ABB RobotStudio station: VRM_Rubik_v12.rspag

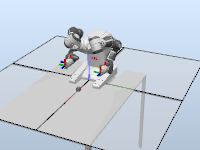
--- station ---
Station VRM_Rubik (saved by RobotStudio 20.4.9280.0)
Controller Controller_Rubik
  mechanical unit ROB_R: IRB14000_0.5_0.5_R, 6 joints, base frame (0, 0, 0) mm
  mechanical unit ROB_R_7: IRB14000_0.5_0.5_R, 1 joints, base frame (0, 0, 0) mm
  mechanical unit ROB_L: IRB14000_0.5_0.5_L, 6 joints, base frame (0, 0, 0) mm
  mechanical unit ROB_L_7: IRB14000_0.5_0.5_L, 1 joints, base frame (0, 0, 0) mm
Layout (positions relative to the parent item):
  - IRB14000_0.5_0.5 [mechanism, from Robots\IRB14000_0.5_0.5__02.rslib] at (0, 0, 0) mm
  - IRB14000_0.5_0.5_R [mechanism, from Robots\IRB14000_0.5_0.5__02.rslib] at (0, 0, 0) mm; joint values [0.0767, -2.326, -2.2629, 0.5469, 0.2972, 1.0609, -0.0992] (rad or m)
  - IRB14000_0.5_0.5_L [mechanism, from Robots\IRB14000_0.5_0.5__02.rslib] at (0, 0, 0) mm; joint values [-0.2847, -2.3545, 2.1434, 0.5675, 2.7327, -0.9321, -2.9148] (rad or m)
  - Smart_Gripper_Servo_Camera_Fingers [mechanism] at (35.8, -200, 200) mm, rotated rx 120.88 ry -90 rz 59.12 deg; joint values [0.025] (rad or m)
      TCP Servo at (0, 0, 114.2) mm
      TCP Camera at (-7.3, 28.3, 35.1) mm, rotated rx 0 ry 90 rz 90 deg
      links: HandBase, DownFinger, UpFinger, VacuumOne, VacuumTwo
  - Smart_Gripper_Servo_Fingers [mechanism] at (35.8, 200, 200) mm, rotated rx 169.62 ry -90 rz 10.38 deg; joint values [0.025] (rad or m)
      TCP Servo at (0, 0, 114.2) mm
      links: HandBase, DownFinger, UpFinger, VacuumOne, VacuumTwo
  - cube_1C3 [part] at (250, -19, 0) mm
  - cube_2C3 [part] at (250, -6, 0) mm
  - cube_3C3 [part] at (250, 7, 0) mm
  - cube_2C2 [part] at (237, -6, 0) mm
  - cube_1C2 [part] at (237, -19, 0) mm
  - cube_3C2 [part] at (237, 7, 0) mm
  - cube_2C1 [part] at (224, -6, 0) mm
  - cube_1C1 [part] at (224, -19, 0) mm
  - cube_3C1 [part] at (224, 7, 0) mm
  - cube_2B1 [part] at (224, -6, 13) mm
  - cube_1B1 [part] at (224, -19, 13) mm
  - cube_3B1 [part] at (224, 7, 13) mm
  - cube_1B2 [part] at (237, -19, 13) mm
  - cube_3B2 [part] at (237, 7, 13) mm
  - cube_2B3 [part] at (250, -6, 13) mm
  - cube_1B3 [part] at (250, -19, 13) mm
  - cube_3B3 [part] at (250, 7, 13) mm
  - core [part] at (243, 0, 19) mm
  - cube_2A3 [part] at (250, -6, 26) mm
  - cube_1A3 [part] at (250, -19, 26) mm
  - cube_3A3 [part] at (250, 7, 26) mm
  - cube_2A2 [part] at (237, -6, 26) mm
  - cube_1A2 [part] at (237, -19, 26) mm
  - cube_3A2 [part] at (237, 7, 26) mm
  - cube_2A1 [part] at (224, -6, 26) mm
  - cube_1A1 [part] at (224, -19, 26) mm
  - cube_3A1 [part] at (224, 7, 26) mm
  - Attacher_3C2 [smart component, from Components\Attacher.rslib]
      properties: Parent=core; Flange=0; Child=cube_3C2; Mount=false; Offset=[0 0 0]; Orientation=[0 0 0]
  - Attacher_1B1 [smart component, from Components\Attacher.rslib]
      properties: Parent=core; Flange=0; Child=cube_1B1; Mount=false; Offset=[0 0 0]; Orientation=[0 0 0]
  - Attacher_1B2 [smart component, from Components\Attacher.rslib]
      properties: Parent=core; Flange=0; Child=cube_1B2; Mount=false; Offset=[0 0 0]; Orientation=[0 0 0]
  - Attacher_1B3 [smart component, from Components\Attacher.rslib]
      properties: Parent=core; Flange=0; Child=cube_1B3; Mount=false; Offset=[0 0 0]; Orientation=[0 0 0]
  - Attacher_1C1 [smart component, from Components\Attacher.rslib]
      properties: Parent=core; Flange=0; Child=cube_1C1; Mount=false; Offset=[0 0 0]; Orientation=[0 0 0]
  - Attacher_1C2 [smart component, from Components\Attacher.rslib]
      properties: Parent=core; Flange=0; Child=cube_1C2; Mount=false; Offset=[0 0 0]; Orientation=[0 0 0]
  - Attacher_1C3 [smart component, from Components\Attacher.rslib]
      properties: Parent=core; Flange=0; Child=cube_1C3; Mount=false; Offset=[0 0 0]; Orientation=[0 0 0]
  - Attacher_2A1 [smart component, from Components\Attacher.rslib]
      properties: Parent=core; Flange=0; Child=cube_2A1; Mount=false; Offset=[0 0 0]; Orientation=[0 0 0]
  - Attacher_2A2 [smart component, from Components\Attacher.rslib]
      properties: Parent=core; Flange=0; Child=cube_2A2; Mount=false; Offset=[0 0 0]; Orientation=[0 0 0]
  - Attacher_2A3 [smart component, from Components\Attacher.rslib]
      properties: Parent=core; Flange=0; Child=cube_2A3; Mount=false; Offset=[0 0 0]; Orientation=[0 0 0]
  - Attacher_2B1 [smart component, from Components\Attacher.rslib]
      properties: Parent=core; Flange=0; Child=cube_2B1; Mount=false; Offset=[0 0 0]; Orientation=[0 0 0]
  - Attacher_2B3 [smart component, from Components\Attacher.rslib]
      properties: Parent=core; Flange=0; Child=cube_2B3; Mount=false; Offset=[0 0 0]; Orientation=[0 0 0]
  - Attacher_2C1 [smart component, from Components\Attacher.rslib]
      properties: Parent=core; Flange=0; Child=cube_2C1; Mount=false; Offset=[0 0 0]; Orientation=[0 0 0]
  - Attacher_2C2 [smart component, from Components\Attacher.rslib]
      properties: Parent=core; Flange=0; Child=cube_2C2; Mount=false; Offset=[0 0 0]; Orientation=[0 0 0]
  - Attacher_2C3 [smart component, from Components\Attacher.rslib]
      properties: Parent=core; Flange=0; Child=cube_2C3; Mount=false; Offset=[0 0 0]; Orientation=[0 0 0]
  - Attacher_3A1 [smart component, from Components\Attacher.rslib]
      properties: Parent=core; Flange=0; Child=cube_3A1; Mount=false; Offset=[0 0 0]; Orientation=[0 0 0]
  - Attacher_3A2 [smart component, from Components\Attacher.rslib]
      properties: Parent=core; Flange=0; Child=cube_3A2; Mount=false; Offset=[0 0 0]; Orientation=[0 0 0]
  - Attacher_3A3 [smart component, from Components\Attacher.rslib]
      properties: Parent=core; Flange=0; Child=cube_3A3; Mount=false; Offset=[0 0 0]; Orientation=[0 0 0]
  - Attacher_3B1 [smart component, from Components\Attacher.rslib]
      properties: Parent=core; Flange=0; Child=cube_3B1; Mount=false; Offset=[0 0 0]; Orientation=[0 0 0]
  - Attacher_3B2 [smart component, from Components\Attacher.rslib]
      properties: Parent=core; Flange=0; Child=cube_3B2; Mount=false; Offset=[0 0 0]; Orientation=[0 0 0]
  - Attacher_3B3 [smart component, from Components\Attacher.rslib]
      properties: Parent=core; Flange=0; Child=cube_3B3; Mount=false; Offset=[0 0 0]; Orientation=[0 0 0]
  - Attacher_3C1 [smart component, from Components\Attacher.rslib]
      properties: Parent=core; Flange=0; Child=cube_3C1; Mount=false; Offset=[0 0 0]; Orientation=[0 0 0]
  - Attacher_3C3 [smart component, from Components\Attacher.rslib]
      properties: Parent=core; Flange=0; Child=cube_3C3; Mount=false; Offset=[0 0 0]; Orientation=[0 0 0]
  - Attacher_1A3 [smart component, from Components\Attacher.rslib]
      properties: Parent=core; Flange=0; Child=cube_1A3; Mount=false; Offset=[0 0 0]; Orientation=[0 0 0]
  - Attacher_1A2 [smart component, from Components\Attacher.rslib]
      properties: Parent=core; Flange=0; Child=cube_1A2; Mount=false; Offset=[0 0 0]; Orientation=[0 0 0]
  - Attacher_1A1 [smart component, from Components\Attacher.rslib]
      properties: Parent=core; Flange=0; Child=cube_1A1; Mount=false; Offset=[0 0 0]; Orientation=[0 0 0]
  - Detacher_1A1 [smart component, from Components\Detacher.rslib]
      properties: Child=cube_1A1; KeepPosition=true
  - Detacher_1A2 [smart component, from Components\Detacher.rslib]
      properties: Child=cube_1A2; KeepPosition=true
  - Detacher_1A3 [smart component, from Components\Detacher.rslib]
      properties: Child=cube_1A3; KeepPosition=true
  - Detacher_1B1 [smart component, from Components\Detacher.rslib]
      properties: Child=cube_1B1; KeepPosition=true
  - Detacher_1B2 [smart component, from Components\Detacher.rslib]
      properties: Child=cube_1B2; KeepPosition=true
  - Detacher_1B3 [smart component, from Components\Detacher.rslib]
      properties: Child=cube_1B3; KeepPosition=true
  - Detacher_1C1 [smart component, from Components\Detacher.rslib]
      properties: Child=cube_1C1; KeepPosition=true
  - Detacher_1C2 [smart component, from Components\Detacher.rslib]
      properties: Child=cube_1C2; KeepPosition=true
  - Detacher_1C3 [smart component, from Components\Detacher.rslib]
      properties: Child=cube_1C3; KeepPosition=true
  - Detacher_2A1 [smart component, from Components\Detacher.rslib]
      properties: Child=cube_2A1; KeepPosition=true
  - Detacher_2A2 [smart component, from Components\Detacher.rslib]
      properties: Child=cube_2A2; KeepPosition=true
  - Detacher_2A3 [smart component, from Components\Detacher.rslib]
      properties: Child=cube_2A3; KeepPosition=true
  - Detacher_2B1 [smart component, from Components\Detacher.rslib]
      properties: Child=cube_2B1; KeepPosition=true
  - Detacher_2B3 [smart component, from Components\Detacher.rslib]
      properties: Child=cube_2B3; KeepPosition=true
  - Detacher_2C1 [smart component, from Components\Detacher.rslib]
      properties: Child=cube_2C1; KeepPosition=true
  - Detacher_2C2 [smart component, from Components\Detacher.rslib]
      properties: Child=cube_2C2; KeepPosition=true
  - Detacher_2C3 [smart component, from Components\Detacher.rslib]
      properties: Child=cube_2C3; KeepPosition=true
  - Detacher_3A1 [smart component, from Components\Detacher.rslib]
      properties: Child=cube_3A1; KeepPosition=true
  - Detacher_3A2 [smart component, from Components\Detacher.rslib]
      properties: Child=cube_3A2; KeepPosition=true
  - Detacher_3A3 [smart component, from Components\Detacher.rslib]
      properties: Child=cube_3A3; KeepPosition=true
  - Detacher_3B1 [smart component, from Components\Detacher.rslib]
      properties: Child=cube_3B1; KeepPosition=true
  - Detacher_3B2 [smart component, from Components\Detacher.rslib]
      properties: Child=cube_3B2; KeepPosition=true
  - Detacher_3B3 [smart component, from Components\Detacher.rslib]
      properties: Child=cube_3B3; KeepPosition=true
  - Detacher_3C1 [smart component, from Components\Detacher.rslib]
      properties: Child=cube_3C1; KeepPosition=true
  - Detacher_3C2 [smart component, from Components\Detacher.rslib]
      properties: Child=cube_3C2; KeepPosition=true
  - Detacher_3C3 [smart component, from Components\Detacher.rslib]
      properties: Child=cube_3C3; KeepPosition=true
  - Positioner_i1A1 [smart component, from Components\Positioner.rslib]
      properties: Object=cube_1A1; Position=[0.224 -0.019 0.026]; Orientation=[0 0 0]; Reference=Global; ReferenceObject=(none)
  - Positioner_i1A2 [smart component, from Components\Positioner.rslib]
      properties: Object=cube_1A2; Position=[0.237 -0.019 0.026]; Orientation=[0 0 0]; Reference=Global; ReferenceObject=(none)
  - Positioner_i1A3 [smart component, from Components\Positioner.rslib]
      properties: Object=cube_1A3; Position=[0.25 -0.019 0.026]; Orientation=[0 0 0]; Reference=Global; ReferenceObject=(none)
  - Positioner_i1B1 [smart component, from Components\Positioner.rslib]
      properties: Object=cube_1B1; Position=[0.224 -0.019 0.013]; Orientation=[0 0 0]; Reference=Global; ReferenceObject=(none)
  - Positioner_i1B2 [smart component, from Components\Positioner.rslib]
      properties: Object=cube_1B2; Position=[0.237 -0.019 0.013]; Orientation=[0 0 0]; Reference=Global; ReferenceObject=(none)
  - Positioner_i1B3 [smart component, from Components\Positioner.rslib]
      properties: Object=cube_1B3; Position=[0.25 -0.019 0.013]; Orientation=[0 0 0]; Reference=Global; ReferenceObject=(none)
  - Positioner_i1C1 [smart component, from Components\Positioner.rslib]
      properties: Object=cube_1C1; Position=[0.224 -0.019 0]; Orientation=[0 0 0]; Reference=Global; ReferenceObject=(none)
  - Positioner_i1C2 [smart component, from Components\Positioner.rslib]
      properties: Object=cube_1C2; Position=[0.237 -0.019 0]; Orientation=[0 0 0]; Reference=Global; ReferenceObject=(none)
  - Positioner_i1C3 [smart component, from Components\Positioner.rslib]
      properties: Object=cube_1C3; Position=[0.25 -0.019 0]; Orientation=[0 0 0]; Reference=Global; ReferenceObject=(none)
  - Positioner_i2A1 [smart component, from Components\Positioner.rslib]
      properties: Object=cube_2A1; Position=[0.224 -0.006 0.026]; Orientation=[0 0 0]; Reference=Global; ReferenceObject=(none)
  - Positioner_i2A2 [smart component, from Components\Positioner.rslib]
      properties: Object=cube_2A2; Position=[0.237 -0.006 0.026]; Orientation=[0 0 0]; Reference=Global; ReferenceObject=(none)
  - Positioner_i2A3 [smart component, from Components\Positioner.rslib]
      properties: Object=cube_2A3; Position=[0.25 -0.006 0.026]; Orientation=[0 0 0]; Reference=Global; ReferenceObject=(none)
  - Positioner_i2B1 [smart component, from Components\Positioner.rslib]
      properties: Object=cube_2B1; Position=[0.224 -0.006 0.013]; Orientation=[0 0 0]; Reference=Global; ReferenceObject=(none)
  - Positioner_i2B3 [smart component, from Components\Positioner.rslib]
      properties: Object=cube_2B3; Position=[0.25 -0.006 0.013]; Orientation=[0 0 0]; Reference=Global; ReferenceObject=(none)
  - Positioner_i2C1 [smart component, from Components\Positioner.rslib]
      properties: Object=cube_2C1; Position=[0.224 -0.006 0]; Orientation=[0 0 0]; Reference=Global; ReferenceObject=(none)
  - Positioner_i2C2 [smart component, from Components\Positioner.rslib]
      properties: Object=cube_2C2; Position=[0.237 -0.006 0]; Orientation=[0 0 0]; Reference=Global; ReferenceObject=(none)
  - Positioner_i2C3 [smart component, from Components\Positioner.rslib]
      properties: Object=cube_2C3; Position=[0.25 -0.006 0]; Orientation=[0 0 0]; Reference=Global; ReferenceObject=(none)
  - Positioner_i3A1 [smart component, from Components\Positioner.rslib]
      properties: Object=cube_3A1; Position=[0.224 0.007 0.026]; Orientation=[0 0 0]; Reference=Global; ReferenceObject=(none)
  - Positioner_i3A2 [smart component, from Components\Positioner.rslib]
      properties: Object=cube_3A2; Position=[0.237 0.007 0.026]; Orientation=[0 0 0]; Reference=Global; ReferenceObject=(none)
  - Positioner_i3A3 [smart component, from Components\Positioner.rslib]
      properties: Object=cube_3A3; Position=[0.25 0.007 0.026]; Orientation=[0 0 0]; Reference=Global; ReferenceObject=(none)
  - Positioner_i3B1 [smart component, from Components\Positioner.rslib]
      properties: Object=cube_3B1; Position=[0.224 0.007 0.013]; Orientation=[0 0 0]; Reference=Global; ReferenceObject=(none)
  - Positioner_i3B2 [smart component, from Components\Positioner.rslib]
      properties: Object=cube_3B2; Position=[0.237 0.007 0.013]; Orientation=[0 0 0]; Reference=Global; ReferenceObject=(none)
  - Positioner_i3B3 [smart component, from Components\Positioner.rslib]
      properties: Object=cube_3B3; Position=[0.25 0.007 0.013]; Orientation=[0 0 0]; Reference=Global; ReferenceObject=(none)
  - Positioner_i3C1 [smart component, from Components\Positioner.rslib]
      properties: Object=cube_3C1; Position=[0.224 0.007 0]; Orientation=[0 0 0]; Reference=Global; ReferenceObject=(none)
  - Positioner_i3C2 [smart component, from Components\Positioner.rslib]
      properties: Object=cube_3C2; Position=[0.237 0.007 0]; Orientation=[0 0 0]; Reference=Global; ReferenceObject=(none)
  - Positioner_i3C3 [smart component, from Components\Positioner.rslib]
      properties: Object=cube_3C3; Position=[0.25 0.007 0]; Orientation=[0 0 0]; Reference=Global; ReferenceObject=(none)
  - Positioner_iCORE [smart component, from Components\Positioner.rslib]
      properties: Object=core; Position=[0.243 0 0.019]; Orientation=[0 0 0]; Reference=Global; ReferenceObject=(none)
  - Positioner_rCORE [smart component, from Components\Positioner.rslib]
      properties: Object=core; Position=[0.25 0 0.2065]; Orientation=[-1.5707963267949 0 0]; Reference=Global; ReferenceObject=(none)
  - Positioner_r1A1 [smart component, from Components\Positioner.rslib] at (231, 7, 225) mm, rotated rx -90 ry 0 rz 0 deg
      properties: Object=cube_1A1; Position=[0.231 0.007 0.2255]; Orientation=[-1.5707963267949 0 0]; Reference=Global; ReferenceObject=(none)
  - Positioner_r1A2 [smart component, from Components\Positioner.rslib] at (244, 7, 225.5) mm, rotated rx -90 ry 0 rz 0 deg
      properties: Object=cube_1A2; Position=[0.244 0.007 0.2255]; Orientation=[-1.5707963267949 0 0]; Reference=Global; ReferenceObject=(none)
  - Positioner_r1A3 [smart component, from Components\Positioner.rslib] at (257, 7, 225.5) mm, rotated rx -90 ry 0 rz 0 deg
      properties: Object=cube_1A3; Position=[0.257 0.007 0.2255]; Orientation=[-1.5707963267949 0 0]; Reference=Global; ReferenceObject=(none)
  - Positioner_r1B1 [smart component, from Components\Positioner.rslib] at (231, -6, 225) mm, rotated rx -90 ry 0 rz 0 deg
      properties: Object=cube_1B1; Position=[0.231 -0.006 0.2255]; Orientation=[-1.5707963267949 0 0]; Reference=Global; ReferenceObject=(none)
  - Positioner_r1B2 [smart component, from Components\Positioner.rslib] at (244, -6, 225.5) mm, rotated rx -90 ry 0 rz 0 deg
      properties: Object=cube_1B2; Position=[0.244 -0.006 0.2255]; Orientation=[-1.5707963267949 0 0]; Reference=Global; ReferenceObject=(none)
  - Positioner_r1B3 [smart component, from Components\Positioner.rslib] at (257, -6, 225.5) mm, rotated rx -90 ry 0 rz 0 deg
      properties: Object=cube_1B3; Position=[0.257 -0.006 0.2255]; Orientation=[-1.5707963267949 0 0]; Reference=Global; ReferenceObject=(none)
  - Positioner_r1C1 [smart component, from Components\Positioner.rslib] at (231, -19, 225.5) mm, rotated rx -90 ry 0 rz 0 deg
      properties: Object=cube_1C1; Position=[0.231 -0.019 0.2255]; Orientation=[-1.5707963267949 0 0]; Reference=Global; ReferenceObject=(none)
  - Positioner_r1C2 [smart component, from Components\Positioner.rslib] at (244, -19, 225.5) mm, rotated rx -90 ry 0 rz 0 deg
      properties: Object=cube_1C2; Position=[0.244 -0.019 0.2255]; Orientation=[-1.5707963267949 0 0]; Reference=Global; ReferenceObject=(none)
  - Positioner_r1C3 [smart component, from Components\Positioner.rslib] at (257, -19, 225.5) mm, rotated rx -90 ry 0 rz 0 deg
      properties: Object=cube_1C3; Position=[0.257 -0.019 0.2255]; Orientation=[-1.5707963267949 0 0]; Reference=Global; ReferenceObject=(none)
  - Positioner_r2A1 [smart component, from Components\Positioner.rslib] at (231, 7, 212.5) mm, rotated rx -90 ry 0 rz 0 deg
      properties: Object=cube_2A1; Position=[0.231 0.007 0.2125]; Orientation=[-1.5707963267949 0 0]; Reference=Global; ReferenceObject=(none)
  - Positioner_r2A2 [smart component, from Components\Positioner.rslib] at (244, 7, 212.5) mm, rotated rx -90 ry 0 rz 0 deg
      properties: Object=cube_2A2; Position=[0.244 0.007 0.2125]; Orientation=[-1.5707963267949 0 0]; Reference=Global; ReferenceObject=(none)
  - Positioner_r2A3 [smart component, from Components\Positioner.rslib] at (257, 7, 212.5) mm, rotated rx -90 ry 0 rz 0 deg
      properties: Object=cube_2A3; Position=[0.257 0.007 0.2125]; Orientation=[-1.5707963267949 0 0]; Reference=Global; ReferenceObject=(none)
  - Positioner_r2B1 [smart component, from Components\Positioner.rslib] at (231, -6, 212.5) mm, rotated rx -90 ry 0 rz 0 deg
      properties: Object=cube_2B1; Position=[0.231 -0.006 0.2125]; Orientation=[-1.5707963267949 0 0]; Reference=Global; ReferenceObject=(none)
  - Positioner_r2B3 [smart component, from Components\Positioner.rslib] at (257, -6, 212.5) mm, rotated rx -90 ry 0 rz 0 deg
      properties: Object=cube_2B3; Position=[0.257 -0.006 0.2125]; Orientation=[-1.5707963267949 0 0]; Reference=Global; ReferenceObject=(none)
  - Positioner_r2C1 [smart component, from Components\Positioner.rslib] at (231, -19, 212.5) mm, rotated rx -90 ry 0 rz 0 deg
      properties: Object=cube_2C1; Position=[0.231 -0.019 0.2125]; Orientation=[-1.5707963267949 0 0]; Reference=Global; ReferenceObject=(none)
  - Positioner_r2C2 [smart component, from Components\Positioner.rslib] at (244, -19, 212.5) mm, rotated rx -90 ry 0 rz 0 deg
      properties: Object=cube_2C2; Position=[0.244 -0.019 0.2125]; Orientation=[-1.5707963267949 0 0]; Reference=Global; ReferenceObject=(none)
  - Positioner_r2C3 [smart component, from Components\Positioner.rslib] at (257, -19, 212.5) mm, rotated rx -90 ry 0 rz 0 deg
      properties: Object=cube_2C3; Position=[0.257 -0.019 0.2125]; Orientation=[-1.5707963267949 0 0]; Reference=Global; ReferenceObject=(none)
  - Positioner_r3A1 [smart component, from Components\Positioner.rslib] at (231, 7, 199.5) mm, rotated rx -90 ry 0 rz 0 deg
      properties: Object=cube_3A1; Position=[0.231 0.007 0.1995]; Orientation=[-1.5707963267949 0 0]; Reference=Global; ReferenceObject=(none)
  - Positioner_r3A2 [smart component, from Components\Positioner.rslib] at (244, 7, 199.5) mm, rotated rx -90 ry 0 rz 0 deg
      properties: Object=cube_3A2; Position=[0.244 0.007 0.1995]; Orientation=[-1.5707963267949 0 0]; Reference=Global; ReferenceObject=(none)
  - Positioner_r3A3 [smart component, from Components\Positioner.rslib] at (257, 7, 199.5) mm, rotated rx -90 ry 0 rz 0 deg
      properties: Object=cube_3A3; Position=[0.257 0.007 0.1995]; Orientation=[-1.5707963267949 0 0]; Reference=Global; ReferenceObject=(none)
  - Positioner_r3B1 [smart component, from Components\Positioner.rslib] at (231, -6, 199.5) mm, rotated rx -90 ry 0 rz 0 deg
      properties: Object=cube_3B1; Position=[0.231 -0.006 0.1995]; Orientation=[-1.5707963267949 0 0]; Reference=Global; ReferenceObject=(none)
  - Positioner_r3B2 [smart component, from Components\Positioner.rslib] at (244, -6, 199.5) mm, rotated rx -90 ry 0 rz 0 deg
      properties: Object=cube_3B2; Position=[0.244 -0.006 0.1995]; Orientation=[-1.5707963267949 0 0]; Reference=Global; ReferenceObject=(none)
  - Positioner_r3B3 [smart component, from Components\Positioner.rslib] at (257, -6, 199.5) mm, rotated rx -90 ry 0 rz 0 deg
      properties: Object=cube_3B3; Position=[0.257 -0.006 0.1995]; Orientation=[-1.5707963267949 0 0]; Reference=Global; ReferenceObject=(none)
  - Positioner_r3C1 [smart component, from Components\Positioner.rslib] at (231, -19, 199.5) mm, rotated rx -90 ry 0 rz 0 deg
      properties: Object=cube_3C1; Position=[0.231 -0.019 0.1995]; Orientation=[-1.5707963267949 0 0]; Reference=Global; ReferenceObject=(none)
  - Positioner_r3C2 [smart component, from Components\Positioner.rslib] at (244, -19, 199.5) mm, rotated rx -90 ry 0 rz 0 deg
      properties: Object=cube_3C2; Position=[0.244 -0.019 0.1995]; Orientation=[-1.5707963267949 0 0]; Reference=Global; ReferenceObject=(none)
  - Positioner_r3C3 [smart component, from Components\Positioner.rslib] at (257, -19, 199.5) mm, rotated rx -90 ry 0 rz 0 deg
      properties: Object=cube_3C3; Position=[0.257 -0.019 0.1995]; Orientation=[-1.5707963267949 0 0]; Reference=Global; ReferenceObject=(none)
  - table [part]
  - Attacher_L [smart component, from Components\Attacher.rslib]
      properties: Parent=Smart_Gripper_Servo_Fingers; Flange=0; Child=core; Mount=false; Offset=[0 0 0]; Orientation=[0 0 0]
  - Attacher_R [smart component, from Components\Attacher.rslib]
      properties: Parent=Smart_Gripper_Servo_Camera_Fingers; Flange=0; Child=core; Mount=false; Offset=[0 0 0]; Orientation=[0 0 0]
  - Detacher_core [smart component, from Components\Detacher.rslib]
      properties: Child=core; KeepPosition=true
Attachment: Smart_Gripper_Servo_Camera_Fingers is attached to IRB14000_0.5_0.5_R / Link7
Attachment: Smart_Gripper_Servo_Fingers is attached to IRB14000_0.5_0.5_L / Link7
EventTableEntry 3147: Group=, Trigger=DO_close_L 3148, Actions=[EventTableActionMechanicalPose 3149], Comment=, ActivationMode=2, Cyclic=false
EventTableTriggerIO 3148: IOValue=[1], IRC5Controller=? -1, Operator=0, SignalSource=Controller_Rubik 1733
EventTableActionMechanicalPose 3149: VirtualSignal=, Mechanism=Smart_Gripper_Servo_Fingers 1554, ToPoseName=SyncPosition, VirtualSignalValue=[1]
EventTableEntry 3164: Group=, Trigger=DO_close_R 3165, Actions=[EventTableActionMechanicalPose 3166], Comment=, ActivationMode=2, Cyclic=false
EventTableTriggerIO 3165: IOValue=[1], IRC5Controller=? -1, Operator=0, SignalSource=Controller_Rubik 1733
EventTableActionMechanicalPose 3166: VirtualSignal=, Mechanism=Smart_Gripper_Servo_Camera_Fingers 1546, ToPoseName=SyncPosition, VirtualSignalValue=[1]
EventTableEntry 3167: Group=, Trigger=DO_open_L 3168, Actions=[EventTableActionMechanicalPose 3169], Comment=, ActivationMode=2, Cyclic=false
EventTableTriggerIO 3168: IOValue=[1], IRC5Controller=? -1, Operator=0, SignalSource=Controller_Rubik 1733
EventTableActionMechanicalPose 3169: VirtualSignal=, Mechanism=Smart_Gripper_Servo_Fingers 1554, ToPoseName=HomePosition, VirtualSignalValue=[1]
EventTableEntry 3170: Group=, Trigger=DO_open_R 3171, Actions=[EventTableActionMechanicalPose 3172], Comment=, ActivationMode=2, Cyclic=false
EventTableTriggerIO 3171: IOValue=[1], IRC5Controller=? -1, Operator=0, SignalSource=Controller_Rubik 1733
EventTableActionMechanicalPose 3172: VirtualSignal=, Mechanism=Smart_Gripper_Servo_Camera_Fingers 1546, ToPoseName=HomePosition, VirtualSignalValue=[1]
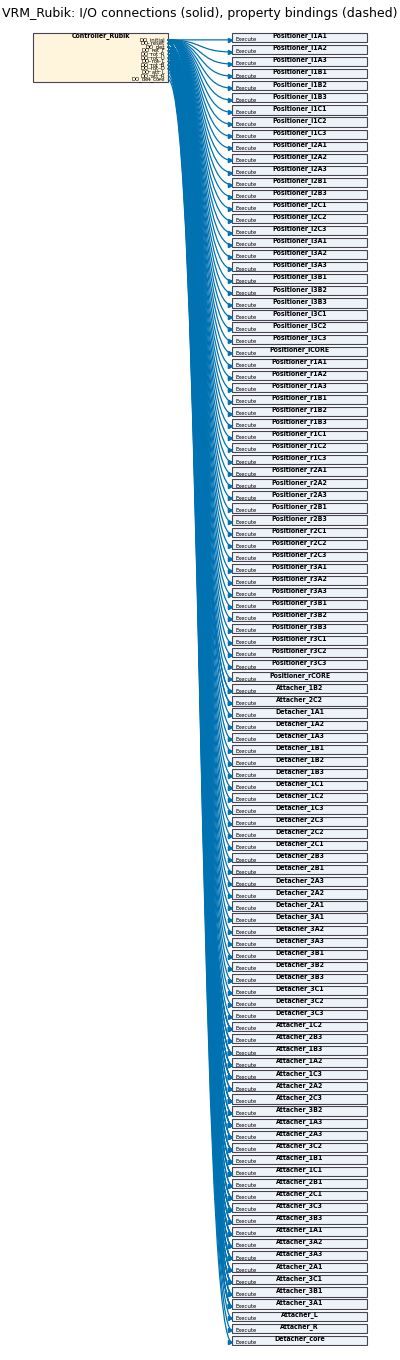
Station logic (signal -> signal, property => property):
  Controller_Rubik.DO_initial -> Positioner_i1A1.Execute
  Controller_Rubik.DO_initial -> Positioner_i1A2.Execute
  Controller_Rubik.DO_initial -> Positioner_i1A3.Execute
  Controller_Rubik.DO_initial -> Positioner_i1B1.Execute
  Controller_Rubik.DO_initial -> Positioner_i1B2.Execute
  Controller_Rubik.DO_initial -> Positioner_i1B3.Execute
  Controller_Rubik.DO_initial -> Positioner_i1C1.Execute
  Controller_Rubik.DO_initial -> Positioner_i1C2.Execute
  Controller_Rubik.DO_initial -> Positioner_i1C3.Execute
  Controller_Rubik.DO_initial -> Positioner_i2A1.Execute
  Controller_Rubik.DO_initial -> Positioner_i2A2.Execute
  Controller_Rubik.DO_initial -> Positioner_i2A3.Execute
  Controller_Rubik.DO_initial -> Positioner_i2B1.Execute
  Controller_Rubik.DO_initial -> Positioner_i2B3.Execute
  Controller_Rubik.DO_initial -> Positioner_i2C1.Execute
  Controller_Rubik.DO_initial -> Positioner_i2C2.Execute
  Controller_Rubik.DO_initial -> Positioner_i2C3.Execute
  Controller_Rubik.DO_initial -> Positioner_i3A1.Execute
  Controller_Rubik.DO_initial -> Positioner_i3A2.Execute
  Controller_Rubik.DO_initial -> Positioner_i3A3.Execute
  Controller_Rubik.DO_initial -> Positioner_i3B1.Execute
  Controller_Rubik.DO_initial -> Positioner_i3B2.Execute
  Controller_Rubik.DO_initial -> Positioner_i3B3.Execute
  Controller_Rubik.DO_initial -> Positioner_i3C1.Execute
  Controller_Rubik.DO_initial -> Positioner_i3C2.Execute
  Controller_Rubik.DO_initial -> Positioner_i3C3.Execute
  Controller_Rubik.DO_initial -> Positioner_iCORE.Execute
  Controller_Rubik.DO_reset -> Positioner_r1A1.Execute
  Controller_Rubik.DO_reset -> Positioner_r1A2.Execute
  Controller_Rubik.DO_reset -> Positioner_r1A3.Execute
  Controller_Rubik.DO_reset -> Positioner_r1B1.Execute
  Controller_Rubik.DO_reset -> Positioner_r1B2.Execute
  Controller_Rubik.DO_reset -> Positioner_r1B3.Execute
  Controller_Rubik.DO_reset -> Positioner_r1C1.Execute
  Controller_Rubik.DO_reset -> Positioner_r1C2.Execute
  Controller_Rubik.DO_reset -> Positioner_r1C3.Execute
  Controller_Rubik.DO_reset -> Positioner_r2A1.Execute
  Controller_Rubik.DO_reset -> Positioner_r2A2.Execute
  Controller_Rubik.DO_reset -> Positioner_r2A3.Execute
  Controller_Rubik.DO_reset -> Positioner_r2B1.Execute
  Controller_Rubik.DO_reset -> Positioner_r2B3.Execute
  Controller_Rubik.DO_reset -> Positioner_r2C1.Execute
  Controller_Rubik.DO_reset -> Positioner_r2C2.Execute
  Controller_Rubik.DO_reset -> Positioner_r2C3.Execute
  Controller_Rubik.DO_reset -> Positioner_r3A1.Execute
  Controller_Rubik.DO_reset -> Positioner_r3A2.Execute
  Controller_Rubik.DO_reset -> Positioner_r3A3.Execute
  Controller_Rubik.DO_reset -> Positioner_r3B1.Execute
  Controller_Rubik.DO_reset -> Positioner_r3B2.Execute
  Controller_Rubik.DO_reset -> Positioner_r3B3.Execute
  Controller_Rubik.DO_reset -> Positioner_r3C1.Execute
  Controller_Rubik.DO_reset -> Positioner_r3C2.Execute
  Controller_Rubik.DO_reset -> Positioner_r3C3.Execute
  Controller_Rubik.DO_reset -> Positioner_rCORE.Execute
  Controller_Rubik.DO_initial -> Attacher_1A1.Execute
  Controller_Rubik.DO_initial -> Attacher_1A2.Execute
  Controller_Rubik.DO_initial -> Attacher_1B1.Execute
  Controller_Rubik.DO_initial -> Attacher_1B2.Execute
  Controller_Rubik.DO_initial -> Attacher_1B3.Execute
  Controller_Rubik.DO_initial -> Attacher_1C1.Execute
  Controller_Rubik.DO_initial -> Attacher_1C2.Execute
  Controller_Rubik.DO_initial -> Attacher_1C3.Execute
  Controller_Rubik.DO_initial -> Attacher_2A1.Execute
  Controller_Rubik.DO_initial -> Attacher_2A2.Execute
  Controller_Rubik.DO_initial -> Attacher_2A3.Execute
  Controller_Rubik.DO_initial -> Attacher_2B1.Execute
  Controller_Rubik.DO_initial -> Attacher_2B3.Execute
  Controller_Rubik.DO_initial -> Attacher_2C1.Execute
  Controller_Rubik.DO_initial -> Attacher_2C2.Execute
  Controller_Rubik.DO_initial -> Attacher_2C3.Execute
  Controller_Rubik.DO_initial -> Attacher_3C3.Execute
  Controller_Rubik.DO_initial -> Attacher_3C2.Execute
  Controller_Rubik.DO_initial -> Attacher_3C1.Execute
  Controller_Rubik.DO_initial -> Attacher_3B3.Execute
  Controller_Rubik.DO_initial -> Attacher_3B2.Execute
  Controller_Rubik.DO_initial -> Attacher_3B1.Execute
  Controller_Rubik.DO_initial -> Attacher_3A3.Execute
  Controller_Rubik.DO_initial -> Attacher_3A2.Execute
  Controller_Rubik.DO_initial -> Attacher_3A1.Execute
  Controller_Rubik.DO_det -> Detacher_1A1.Execute
  Controller_Rubik.DO_det -> Detacher_1A2.Execute
  Controller_Rubik.DO_det -> Detacher_1A3.Execute
  Controller_Rubik.DO_det -> Detacher_1B1.Execute
  Controller_Rubik.DO_det -> Detacher_1B2.Execute
  Controller_Rubik.DO_det -> Detacher_1B3.Execute
  Controller_Rubik.DO_det -> Detacher_1C1.Execute
  Controller_Rubik.DO_det -> Detacher_1C2.Execute
  Controller_Rubik.DO_det -> Detacher_1C3.Execute
  Controller_Rubik.DO_det -> Detacher_2C3.Execute
  Controller_Rubik.DO_det -> Detacher_2C2.Execute
  Controller_Rubik.DO_det -> Detacher_2C1.Execute
  Controller_Rubik.DO_det -> Detacher_2B3.Execute
  Controller_Rubik.DO_det -> Detacher_2B1.Execute
  Controller_Rubik.DO_det -> Detacher_2A3.Execute
  Controller_Rubik.DO_det -> Detacher_2A2.Execute
  Controller_Rubik.DO_det -> Detacher_2A1.Execute
  Controller_Rubik.DO_det -> Detacher_3A1.Execute
  Controller_Rubik.DO_det -> Detacher_3A2.Execute
  Controller_Rubik.DO_det -> Detacher_3A3.Execute
  Controller_Rubik.DO_det -> Detacher_3B1.Execute
  Controller_Rubik.DO_det -> Detacher_3B2.Execute
  Controller_Rubik.DO_det -> Detacher_3B3.Execute
  Controller_Rubik.DO_det -> Detacher_3C1.Execute
  Controller_Rubik.DO_det -> Detacher_3C2.Execute
  Controller_Rubik.DO_det -> Detacher_3C3.Execute
  Controller_Rubik.DO_rot_F -> Attacher_1A1.Execute
  Controller_Rubik.DO_rot_F -> Attacher_1A2.Execute
  Controller_Rubik.DO_rot_F -> Attacher_1A3.Execute
  Controller_Rubik.DO_initial -> Attacher_1A3.Execute
  Controller_Rubik.DO_rot_F -> Attacher_1B1.Execute
  Controller_Rubik.DO_rot_F -> Attacher_1B2.Execute
  Controller_Rubik.DO_rot_F -> Attacher_1B3.Execute
  Controller_Rubik.DO_rot_F -> Attacher_1C1.Execute
  Controller_Rubik.DO_rot_F -> Attacher_1C2.Execute
  Controller_Rubik.DO_rot_F -> Attacher_1C3.Execute
  Controller_Rubik.DO_rot_R -> Attacher_1C1.Execute
  Controller_Rubik.DO_rot_R -> Attacher_1C2.Execute
  Controller_Rubik.DO_rot_R -> Attacher_1C3.Execute
  Controller_Rubik.DO_rot_R -> Attacher_2C1.Execute
  Controller_Rubik.DO_rot_R -> Attacher_2C2.Execute
  Controller_Rubik.DO_rot_R -> Attacher_2C3.Execute
  Controller_Rubik.DO_rot_R -> Attacher_3C1.Execute
  Controller_Rubik.DO_rot_R -> Attacher_3C2.Execute
  Controller_Rubik.DO_rot_R -> Attacher_3C3.Execute
  Controller_Rubik.DO_rot_U -> Attacher_1A3.Execute
  Controller_Rubik.DO_rot_U -> Attacher_1B3.Execute
  Controller_Rubik.DO_rot_U -> Attacher_1C3.Execute
  Controller_Rubik.DO_rot_U -> Attacher_2C3.Execute
  Controller_Rubik.DO_rot_U -> Attacher_2B3.Execute
  Controller_Rubik.DO_rot_U -> Attacher_2A3.Execute
  Controller_Rubik.DO_rot_U -> Attacher_3A3.Execute
  Controller_Rubik.DO_rot_U -> Attacher_3B3.Execute
  Controller_Rubik.DO_rot_U -> Attacher_3C3.Execute
  Controller_Rubik.DO_rot_L -> Attacher_1A1.Execute
  Controller_Rubik.DO_rot_L -> Attacher_1A2.Execute
  Controller_Rubik.DO_rot_L -> Attacher_1A3.Execute
  Controller_Rubik.DO_rot_L -> Attacher_2A1.Execute
  Controller_Rubik.DO_rot_L -> Attacher_2A2.Execute
  Controller_Rubik.DO_rot_L -> Attacher_2A3.Execute
  Controller_Rubik.DO_rot_L -> Attacher_3A1.Execute
  Controller_Rubik.DO_rot_L -> Attacher_3A2.Execute
  Controller_Rubik.DO_rot_L -> Attacher_3A3.Execute
  Controller_Rubik.DO_rot_B -> Attacher_3A1.Execute
  Controller_Rubik.DO_rot_B -> Attacher_3A2.Execute
  Controller_Rubik.DO_rot_B -> Attacher_3A3.Execute
  Controller_Rubik.DO_rot_B -> Attacher_3B1.Execute
  Controller_Rubik.DO_rot_B -> Attacher_3B2.Execute
  Controller_Rubik.DO_rot_B -> Attacher_3B3.Execute
  Controller_Rubik.DO_rot_B -> Attacher_3C1.Execute
  Controller_Rubik.DO_rot_B -> Attacher_3C2.Execute
  Controller_Rubik.DO_rot_B -> Attacher_3C3.Execute
  Controller_Rubik.DO_rot_D -> Attacher_1A1.Execute
  Controller_Rubik.DO_rot_D -> Attacher_2A1.Execute
  Controller_Rubik.DO_rot_D -> Attacher_3A1.Execute
  Controller_Rubik.DO_rot_D -> Attacher_1B1.Execute
  Controller_Rubik.DO_rot_D -> Attacher_2B1.Execute
  Controller_Rubik.DO_rot_D -> Attacher_3B1.Execute
  Controller_Rubik.DO_rot_D -> Attacher_1C1.Execute
  Controller_Rubik.DO_rot_D -> Attacher_2C1.Execute
  Controller_Rubik.DO_rot_D -> Attacher_3C1.Execute
  Controller_Rubik.DO_att_L -> Attacher_L.Execute
  Controller_Rubik.DO_att_R -> Attacher_R.Execute
  Controller_Rubik.DO_det_core -> Detacher_core.Execute
Targets, tools, work objects and paths stored in the station and not in the controller backup, written as RAPID:
! task T_ROB_R
MODULE Module1
  PROC Path_camera()
    MoveL Target_F_1,v1000,z100,Servo\WObj:=wobj0;
    MoveL Target_waiting,v1000,z100,Servo\WObj:=wobj0;
    MoveL Target_10,v1000,z100,Servo\WObj:=wobj0;
    MoveL Target_20,v1000,z100,Servo\WObj:=wobj0;
    MoveL Target_30,v1000,z100,Servo\WObj:=wobj0;
    MoveL Target_40,v1000,z100,Servo\WObj:=wobj0;
    MoveL Target_50,v1000,z100,Servo\WObj:=wobj0;
    MoveL Target_60,v1000,z100,Servo\WObj:=wobj0;
    MoveL Target_F,v1000,z100,Servo\WObj:=wobj0;
    MoveL Target_F_rot,v1000,z100,Servo\WObj:=wobj0;
    MoveL Target_home,v1000,z100,Servo\WObj:=wobj0;
    MoveL Target_R,v1000,z100,Servo\WObj:=wobj0;
    MoveL Target_R_rot,v1000,z100,Servo\WObj:=wobj0;
    MoveJ Target_home,v100,fine,Servo\WObj:=wobj0;
    MoveL Target_10,v100,fine,Servo\WObj:=wobj0;
    MoveJ Target_20,v100,fine,Servo\WObj:=wobj0;
    MoveL Target_30,v100,fine,Servo\WObj:=wobj0;
    MoveL Target_40,v100,fine,Servo\WObj:=wobj0;
    MoveL Target_50,v100,fine,Servo\WObj:=wobj0;
    MoveJ Target_60,v100,fine,Servo\WObj:=wobj0;
    MoveL Target_home,v100,fine,Servo\WObj:=wobj0;
    MoveL Target_F_1,v1000,z100,Servo\WObj:=wobj0;
    MoveL Target_F_1rot,v1000,z100,Servo\WObj:=wobj0;
    MoveL Target_B,v1000,z100,Servo\WObj:=wobj0;
    MoveL Target_D,v1000,z100,Servo\WObj:=wobj0;
    MoveL Target_U,v1000,z100,Servo\WObj:=wobj0;
  ENDPROC
ENDMODULE

! task T_ROB_L
MODULE Module1
  PROC Path_pick_up()
    MoveJ Target_10,v100,z100,Servo\WObj:=wobj0;
    MoveJ Target_20,v100,fine,Servo\WObj:=wobj0;
    MoveJ Target_waiting,v100,fine,Servo\WObj:=wobj0;
    MoveL Target_L,v1000,z100,Servo\WObj:=wobj0;
    MoveL Target_L_rot,v1000,z100,Servo\WObj:=wobj0;
    MoveL Target_B,v1000,z100,Servo\WObj:=wobj0;
    MoveL Target_B_rot,v1000,z100,Servo\WObj:=wobj0;
    MoveL Target_D,v1000,z100,Servo\WObj:=wobj0;
    MoveL Target_D_rot,v1000,z100,Servo\WObj:=wobj0;
    MoveL Target_U,v1000,z100,Servo\WObj:=wobj0;
    MoveL Target_U_rot,v1000,z100,Servo\WObj:=wobj0;
  ENDPROC
ENDMODULE


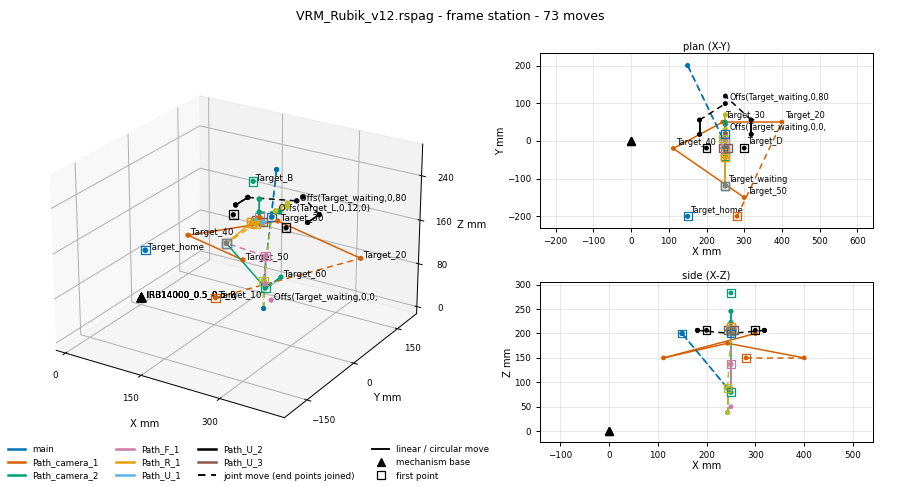
[picture p0: tool path of VRM_Rubik_v12.rspag in frame station, 73 of 73 moves have a stored position in this frame; points joined in program order, loops and branches not executed]
--- Backups/Controller_Rubik/RAPID/TASK1/PROGMOD/CalibData.mod ---
MODULE CalibData
    PERS tooldata Servo:=[TRUE,[[0,0,114.2],[1,0,0,0]],[0.229,[7.9,12.4,48.7],[1,0,0,0],0.00021,0.00023,0.00008]];
    PERS tooldata Camera:=[TRUE,[[-7.3,28.3,35.1],[0.5,-0.5,0.5,0.5]],[0.229,[7.9,12.4,48.7],[1,0,0,0],0.00021,0.00023,0.00008]];
ENDMODULE

--- Backups/Controller_Rubik/RAPID/TASK1/PROGMOD/Module1.mod ---
MODULE Module1
    CONST robtarget Target_10:=[[281,-200,150],[0.683012702,-0.183012702,0.683012702,-0.183012702],[0,0,1,4],[-101.964427132,9E+09,9E+09,9E+09,9E+09,9E+09]];
    CONST robtarget Target_20:=[[400,50,150],[0.612372436,-0.612372436,0.353553391,0.353553391],[1,-1,-1,4],[-101.964427132,9E+09,9E+09,9E+09,9E+09,9E+09]];
    CONST robtarget Target_30:=[[243,50,180],[0.707106781,-0.707106781,0,0],[1,-1,2,4],[-101.964427132,9E+09,9E+09,9E+09,9E+09,9E+09]];
    CONST robtarget Target_40:=[[112,-20,150],[0.612372436,-0.612372436,-0.353553391,-0.353553391],[0,-1,1,4],[-101.964427132,9E+09,9E+09,9E+09,9E+09,9E+09]];
    CONST robtarget Target_50:=[[300,-150,200],[0.707106781,0,0.707106781,0],[0,1,2,4],[-101.964427132,9E+09,9E+09,9E+09,9E+09,9E+09]];
    CONST robtarget Target_60:=[[250,50,80],[0,0,0.707106781,0.707106781],[1,-1,0,4],[-101.964427132,9E+09,9E+09,9E+09,9E+09,9E+09]];
    CONST robtarget Target_home:=[[150,-200,200],[0,0.707106781,0,0.707106781],[0,0,0,4],[-101.964427132,9E+09,9E+09,9E+09,9E+09,9E+09]];
    CONST robtarget Target_F:=[[250,0,225.5],[0,1,0,0],[-1,1,1,1],[-101.964421054,9E+09,9E+09,9E+09,9E+09,9E+09]];
    CONST robtarget Target_F_rot:=[[250,0,225.5],[0,-0.707106781,0.707106781,0],[-1,1,-2,1],[-101.964421054,9E+09,9E+09,9E+09,9E+09,9E+09]];
    CONST robtarget Target_R:=[[250,-19,206.5],[0.5,-0.5,-0.5,-0.5],[1,-1,1,4],[-101.964421054,9E+09,9E+09,9E+09,9E+09,9E+09]];
    CONST robtarget Target_R_rot:=[[250,-19,206.5],[0.707106781,-0.707106781,0,0],[1,-1,2,4],[-101.964421054,9E+09,9E+09,9E+09,9E+09,9E+09]];
    CONST robtarget Target_waiting:=[[250,-119,205],[0.5,-0.5,-0.5,-0.5],[1,-1,1,4],[-101.964421054,9E+09,9E+09,9E+09,9E+09,9E+09]];
    CONST robtarget Target_F_1:=[[250,0,75.5],[0,1,0,0],[1,2,-2,4],[-101.964421054,9E+09,9E+09,9E+09,9E+09,9E+09]];
    CONST robtarget Target_F_1rot:=[[250,0,75.5],[0,-0.707106781,0.707106781,0],[1,2,-1,4],[-101.964421054,9E+09,9E+09,9E+09,9E+09,9E+09]];
    CONST robtarget Target_B:=[[250,-39,283],[0.707106781,-0.707106781,0,0],[1,-1,-2,4],[-101.964421054,9E+09,9E+09,9E+09,9E+09,9E+09]];
    CONST robtarget Target_D:=[[300,-19,206.5],[0,0.707106781,0,0.707106781],[1,1,-1,4],[-101.964421054,9E+09,9E+09,9E+09,9E+09,9E+09]];
    CONST robtarget Target_U:=[[200,-19,206.5],[0.707106781,0,-0.707106781,0],[1,-1,1,4],[-101.964421054,9E+09,9E+09,9E+09,9E+09,9E+09]];

    PERS num state;
    PERS bool sync;
    VAR num state_R := 0;
    VAR socketdev serverSocket;
    VAR socketdev clientSocket;
    VAR string data;
    VAR string actualMove;
    VAR string dictionaryStr := "xxFRULBD";
    VAR num stringLen := 0;
    VAR num pos;

    PROC main()
        TEST state_R
            CASE 0: ! initial
                state := 2;
                Reset DO_rdy_L;
                Reset DO_rdy_R;
                PulseDO DO_det;
                PulseDO DO_det_core;
                PulseDO DO_initial;
                PulseDO DO_open_R;
                MoveJ Target_home,v100,fine,Servo\WObj:=wobj0;
                Path_camera_1;
                PulseDO DO_rdy_R;
                WaitDO DO_rdy_L, 1;
                Path_camera_2;
                PulseDO DO_rdy_R;
                state_R := 1;

            CASE 1: ! waiting for data
                SocketCreate serverSocket;
                SocketBind serverSocket, "127.0.0.1", 31254;
                SocketListen serverSocket;

                SocketAccept serverSocket, clientSocket, \Time:=WAIT_MAX;

                SocketReceive clientSocket \Str:=data;
                SocketSend clientSocket \Str:="recieved";

                SocketClose clientSocket;
                SocketClose serverSocket;

                stringLen := StrLen(data);

                IF stringLen <> 0  THEN
                    state_R := 2;
                ENDIF

            CASE 2: ! next move
                IF StrLen(data) = 0 THEN
                    WaitTime 2;
		            state := 10;
                    state_R := 10;
                ELSE
                    actualMove := StrPart(data, 1, 1);
                    data := StrPart(data, 2, stringLen-1);
                    stringLen := StrLen(data);
                    pos := StrFind(dictionaryStr, 1, actualMove);
		            state := pos;
                    state_R := pos;
                ENDIF

            CASE 3: ! F
                state := 9;
                WaitDO DO_rdy_L, 1;
                Path_F_1;
                PulseDO DO_rdy_R;
                state_R := 31;

            CASE 31:
                WaitDO DO_rdy_L, 1;
                state_R := 9;

            CASE 4: ! R
                state := 9;
                Path_R_1;
                PulseDO DO_rdy_R;
                state_R := 9;

            CASE 5: ! U
                state := 9;
                Path_U_1;
                PulseDO DO_rdy_R;
                state_R := 51;

            CASE 51:
                WaitDO DO_rdy_L, 1;
                Path_U_2;
                PulseDO DO_rdy_R;
                state_R := 52;

            CASE 52:
                WaitDO DO_rdy_L, 1;
                Path_U_3;
                PulseDO DO_rdy_R;
                state_R := 53;

            CASE 53:
                WaitDO DO_rdy_L, 1;
                Path_U_4;
                PulseDO DO_rdy_R;
                state_R := 9;

            CASE 6: ! L
                state := 9;
                Path_L_1;
                PulseDO DO_rdy_R;
                state_R := 61;

            CASE 61:
                WaitDO DO_rdy_L, 1;
                Path_L_2;
                state_R := 9;

            CASE 7: ! B
                state := 9;
                Path_B_1;
                PulseDO DO_rdy_R;
                state_R := 71;

            CASE 71:
                WaitDO DO_rdy_L, 1;
                Path_B_2;
                PulseDO DO_rdy_R;
                state_R := 72;

            CASE 72:
                WaitDO DO_rdy_L, 1;
                Path_B_3;
                PulseDO DO_rdy_R;
                state_R := 73;

            CASE 73:
                WaitDO DO_rdy_L, 1;
                Path_B_4;
                state_R := 9;

            CASE 8: ! D
                state := 9;
                Path_D_1;
                PulseDO DO_rdy_R;
                state_R := 81;

            CASE 81:
                WaitDO DO_rdy_L, 1;
                Path_D_2;
                PulseDO DO_rdy_R;
                state_R := 82;

            CASE 82:
                WaitDO DO_rdy_L, 1;
                Path_D_3;
                PulseDO DO_rdy_R;
                state_R := 83;

            CASE 83:
                WaitDO DO_rdy_L, 1;
                Path_D_4;
                PulseDO DO_rdy_R;
                state_R := 9;

            CASE 9:
                IF sync = TRUE THEN
                    state := 2;
                    state_R := 2;
                ENDIF

            CASE 10: ! end
                MoveJ Target_home,v100,fine,Servo\WObj:=wobj0;
                PulseDO DO_rdy_R;
        ENDTEST
    ENDPROC

    PROC Path_camera_1()
        MoveL Target_10,v100,fine,Servo\WObj:=wobj0;
        WaitTime 0.5;
        MoveJ Target_20,v100,fine,Servo\WObj:=wobj0;
        WaitTime 0.5;
        MoveL Target_30,v100,fine,Servo\WObj:=wobj0;
        WaitTime 0.5;
        MoveL Target_40,v100,fine,Servo\WObj:=wobj0;
        WaitTime 0.5;
        MoveL Target_50,v100,fine,Servo\WObj:=wobj0;
    ENDPROC

    PROC Path_camera_2()
        WaitTime 1;
        MoveJ Offs(Target_60, 0, -50, 0),v100,fine,Servo;
        MoveJ Target_60,v100,fine,Servo\WObj:=wobj0;
        WaitTime 0.5;
        MoveJ Offs(Target_60, 0, -50, 0),v100,fine,Servo;
        MoveL Target_waiting,v100,fine,Servo\WObj:=wobj0;
    ENDPROC

    PROC Path_F_1()
        MoveJ Offs(Target_F_1, 0, 0, 62),v100,z100,Servo;
        MoveL Offs(Target_F_1, 0, 0, 12),v100,fine,Servo;
        WaitTime 1;
        PulseDO DO_close_R;
        WaitTime 1;
        PulseDO DO_att_R;
        PulseDO DO_rot_F;
        MoveJ Offs(Target_F_1rot, 0, 0, 12),v100,fine,Servo;
        PulseDO DO_det;
        PulseDO DO_det_core;
        WaitTime 1;
        PulseDO DO_open_R;
        WaitTime 1;
        MoveJ Offs(Target_F_1rot, 0, 0, 62),v100,z100,Servo;
        MoveJ Target_waiting,v100,fine,Servo\WObj:=wobj0;
    ENDPROC

    PROC Path_R_1()
        MoveL Offs(Target_R, 0, -12, 0),v100,fine,Servo;
        WaitTime 1;
        PulseDO DO_close_R;
        WaitTime 1;
        PulseDO DO_att_R;
        PulseDO DO_rot_R;
        MoveJ Offs(Target_R_rot, 0, -12, 0),v100,fine,Servo;
        PulseDO DO_det;
        PulseDO DO_det_core;
        PulseDO DO_reset;
        WaitTime 1;
        PulseDO DO_open_R;
        WaitTime 1;
        MoveJ Target_waiting,v100,fine,Servo\WObj:=wobj0;
    ENDPROC

    PROC Path_U_1()
        MoveL Offs(Target_R, -6.5, 0, 0),v100,fine,Servo;
        WaitTime 1;
        PulseDO DO_close_R;
        WaitTime 1;
        PulseDO DO_att_R;
        PulseDO DO_rot_F;
        PulseDO DO_rot_R;
        PulseDO DO_rot_U;
        PulseDO DO_rot_L;
        PulseDO DO_rot_B;
        PulseDO DO_rot_D;
    ENDPROC

    PROC Path_U_2()
        MoveJ Target_U,v100,fine,Servo\WObj:=wobj0;
        PulseDO DO_det;
        PulseDO DO_det_core;
    ENDPROC

    PROC Path_U_3()
        PulseDO DO_att_R;
        PulseDO DO_rot_F;
        PulseDO DO_rot_R;
        PulseDO DO_rot_U;
        PulseDO DO_rot_L;
        PulseDO DO_rot_B;
        PulseDO DO_rot_D;
        MoveJ Offs(Target_R, -6.5, 0, 0),v100,fine,Servo;
        PulseDO DO_det;
        PulseDO DO_det_core;
        PulseDO DO_reset;
    ENDPROC

    PROC Path_U_4()
        WaitTime 3;
        PulseDO DO_open_R;
        WaitTime 1;
        MoveL Target_waiting,v100,fine,Servo\WObj:=wobj0;
    ENDPROC

    PROC Path_L_1()
        MoveL Target_R,v100,fine,Servo\WObj:=wobj0;
        WaitTime 1;
        PulseDO DO_close_R;
        WaitTime 1;
    ENDPROC

    PROC Path_L_2()
        WaitTime 1;
        PulseDO DO_open_R;
        WaitTime 1;
        MoveL Target_waiting,v100,fine,Servo\WObj:=wobj0;
    ENDPROC

    PROC Path_B_1()
        MoveL Offs(Target_R_rot, 0, -25, 6.5),v100,z100,Servo;
        MoveL Offs(Target_R_rot, 0, 0, 6.5),v100,fine,Servo;
        WaitTime 1;
        PulseDO DO_close_R;
        WaitTime 1;
        PulseDO DO_att_R;
        PulseDO DO_rot_F;
        PulseDO DO_rot_R;
        PulseDO DO_rot_U;
        PulseDO DO_rot_L;
        PulseDO DO_rot_B;
        PulseDO DO_rot_D;
    ENDPROC

    PROC Path_B_2()
        MoveJ Target_B,v100,fine,Servo\WObj:=wobj0;
        PulseDO DO_det;
        PulseDO DO_det_core;
    ENDPROC

    PROC Path_B_3()
        PulseDO DO_att_R;
        PulseDO DO_rot_F;
        PulseDO DO_rot_R;
        PulseDO DO_rot_U;
        PulseDO DO_rot_L;
        PulseDO DO_rot_B;
        PulseDO DO_rot_D;
        MoveJ Offs(Target_R_rot, 0, 0, 6.5),v100,fine,Servo;
        PulseDO DO_det;
        PulseDO DO_det_core;
        PulseDO DO_reset;
    ENDPROC

    PROC Path_B_4()
        WaitTime 1;
        PulseDO DO_open_R;
        WaitTime 1;
        MoveL Offs(Target_R_rot, 0, -25, 6.5),v100,z100,Servo;
        MoveL Target_waiting,v100,fine,Servo\WObj:=wobj0;
    ENDPROC

    PROC Path_D_1()
        MoveL Offs(Target_R, 6.5, 0, 0),v100,fine,Servo;
        WaitTime 1;
        PulseDO DO_close_R;
        WaitTime 1;
        PulseDO DO_att_R;
        PulseDO DO_rot_F;
        PulseDO DO_rot_R;
        PulseDO DO_rot_U;
        PulseDO DO_rot_L;
        PulseDO DO_rot_B;
        PulseDO DO_rot_D;
    ENDPROC

    PROC Path_D_2()
        MoveJ Target_D,v100,fine,Servo\WObj:=wobj0;
        PulseDO DO_det;
        PulseDO DO_det_core;
    ENDPROC

    PROC Path_D_3()
        PulseDO DO_att_R;
        PulseDO DO_rot_F;
        PulseDO DO_rot_R;
        PulseDO DO_rot_U;
        PulseDO DO_rot_L;
        PulseDO DO_rot_B;
        PulseDO DO_rot_D;
        MoveJ Offs(Target_R, 6.5, 0, 0),v100,fine,Servo;
        PulseDO DO_det;
        PulseDO DO_det_core;
        PulseDO DO_reset;
    ENDPROC

    PROC Path_D_4()
        WaitTime 1;
        PulseDO DO_open_R;
        WaitTime 1;
        MoveL Target_waiting,v100,fine,Servo\WObj:=wobj0;
    ENDPROC
ENDMODULE

--- Backups/Controller_Rubik/RAPID/TASK2/PROGMOD/CalibData.mod ---
MODULE CalibData
    PERS tooldata Servo:=[TRUE,[[0,0,114.2],[1,0,0,0]],[0.215,[8.7,12.3,49.2],[1,0,0,0],0.00021,0.00024,0.00009]];
ENDMODULE

--- Backups/Controller_Rubik/RAPID/TASK2/PROGMOD/Module1.mod ---
MODULE Module1
    CONST robtarget Target_10:=[[243,6.5,88],[0,1,0,0],[-1,-2,2,4],[101.964427132,9E+09,9E+09,9E+09,9E+09,9E+09]];
    CONST robtarget Target_20:=[[243,6.5,38],[0,1,0,0],[-1,-2,2,4],[101.964427132,9E+09,9E+09,9E+09,9E+09,9E+09]];
    CONST robtarget Target_waiting:=[[250,19,200],[0.707106781,0.707106781,0,0],[-1,1,-2,4],[101.964427132,9E+09,9E+09,9E+09,9E+09,9E+09]];
    CONST robtarget Target_home:=[[150,200,200],[0,0.707106781,0,0.707106781],[0,2,-2,5],[105.931421002,9E+09,9E+09,9E+09,9E+09,9E+09]];
    CONST robtarget Target_L:=[[250,19,206.5],[0.707106781,0.707106781,0,0],[-1,1,-2,4],[101.964427132,9E+09,9E+09,9E+09,9E+09,9E+09]];
    CONST robtarget Target_L_rot:=[[250,19,206.5],[0.5,0.5,-0.5,0.5],[-1,1,-2,4],[101.964427132,9E+09,9E+09,9E+09,9E+09,9E+09]];
    CONST robtarget Target_B:=[[250,-20,257.5],[0,0,0,1],[-1,0,0,4],[105.490331729,9E+09,9E+09,9E+09,9E+09,9E+09]];
    CONST robtarget Target_B_rot:=[[250,-20,257.5],[0.707106781,0,0,-0.707106781],[-1,0,0,4],[105.490331729,9E+09,9E+09,9E+09,9E+09,9E+09]];
    CONST robtarget Target_D:=[[318.5,5.5,206.5],[0.5,0.5,-0.5,0.5],[-1,1,-1,4],[101.964427132,9E+09,9E+09,9E+09,9E+09,9E+09]];
    CONST robtarget Target_D_rot:=[[318.5,5.5,206.5],[0,0,-0.707106781,0.707106781],[-1,1,-1,4],[101.964427132,9E+09,9E+09,9E+09,9E+09,9E+09]];
    CONST robtarget Target_U:=[[181.5,5.5,206.5],[0.5,0.5,-0.5,0.5],[0,1,-1,4],[105.931418404,9E+09,9E+09,9E+09,9E+09,9E+09]];
    CONST robtarget Target_U_rot:=[[181.5,5.5,206.5],[0,0,-0.707106781,0.707106781],[0,1,-1,4],[105.931418404,9E+09,9E+09,9E+09,9E+09,9E+09]];

    PERS num state;
    PERS bool sync;
    VAR num state_L := 0;

    PROC main()
        TEST state_L
            CASE 0: ! initial
                Reset DO_rdy_L;
                Reset DO_rdy_R;
                PulseDO DO_open_L;
                MoveJ Target_home,v100,fine,Servo\WObj:=wobj0;
                WaitDO DO_rdy_R, 1;
                Path_pick_up_1;
                PulseDO DO_rdy_L;
                WaitDO DO_rdy_R, 1;
                state_L := 2;

            CASE 2: ! next move
                sync := FALSE;
                state_L := state;

            CASE 3: ! F
                Path_F_1;
                PulseDO DO_rdy_L;
                state_L := 31;

            CASE 31:
                WaitDO DO_rdy_R, 1;
                Path_F_2;
                PulseDO DO_rdy_L;
                state_L := 2;

            CASE 4: ! R
                WaitDO DO_rdy_R, 1;
                state_L := 2;

            CASE 5: ! U
                WaitDO DO_rdy_R, 1;
                Path_U_1;
                PulseDO DO_rdy_L;
                state_L := 51;

            CASE 51:
                WaitDO DO_rdy_R, 1;
                Path_U_2;
                PulseDO DO_rdy_L;
                state_L := 52;

            CASE 52:
                WaitDO DO_rdy_R, 1;
                Path_U_3;
                PulseDO DO_rdy_L;
                state_L := 2;

            CASE 6: ! L
                WaitDO DO_rdy_R, 1;
                Path_L_1;
                PulseDO DO_rdy_L;
                state_L := 2;

            CASE 7: ! B
                WaitDO DO_rdy_R, 1;
                Path_B_1;
                PulseDO DO_rdy_L;
                state_L := 71;

            CASE 71:
                WaitDO DO_rdy_R, 1;
                Path_B_2;
                PulseDO DO_rdy_L;
                state_L := 72;

            CASE 72:
                WaitDO DO_rdy_R, 1;
                Path_B_3;
                PulseDO DO_rdy_L;
                state_L := 2;

            CASE 8: ! D
                WaitDO DO_rdy_R, 1;
                Path_D_1;
                PulseDO DO_rdy_L;
                state_L := 81;

            CASE 81:
                WaitDO DO_rdy_R, 1;
                Path_D_2;
                PulseDO DO_rdy_L;
                state_L := 82;

            CASE 82:
                WaitDO DO_rdy_R, 1;
                Path_D_3;
                PulseDO DO_rdy_L;
                state_L := 2;

            CASE 9:
                sync := TRUE;
                state_L := state;

            CASE 10: ! end
                WaitDO DO_rdy_R, 1;
                PulseDO DO_att_L;
                PulseDO DO_rot_F;
                PulseDO DO_rot_R;
                PulseDO DO_rot_U;
                PulseDO DO_rot_L;
                PulseDO DO_rot_B;
                PulseDO DO_rot_D;
                MoveJ Target_10,v100,z100,Servo\WObj:=wobj0;
                MoveJ Target_20,v100,fine,Servo\WObj:=wobj0;
                PulseDO DO_det;
                PulseDO DO_det_core;
                WaitTime 1;
                PulseDO DO_open_L;
                WaitTime 1;
                MoveJ Target_10,v100,z100,Servo\WObj:=wobj0;
                MoveJ Target_home,v100,fine,Servo\WObj:=wobj0;
                EXIT;
        ENDTEST
    ENDPROC

    PROC Path_pick_up_1()
        MoveJ Target_10,v100,z100,Servo\WObj:=wobj0;
        MoveJ Target_20,v100,fine,Servo\WObj:=wobj0;
        PulseDO DO_att_L;
        WaitTime 1;
        PulseDO DO_close_L;
        WaitTime 1;
        MoveJ Target_10,v100,z100,Servo\WObj:=wobj0;
        MoveJ Target_waiting,v100,fine,Servo\WObj:=wobj0;
        PulseDO DO_det;
        PulseDO DO_det_core;
    ENDPROC

    PROC Path_F_1()
        PulseDO DO_att_L;
        PulseDO DO_rot_F;
        PulseDO DO_rot_R;
        PulseDO DO_rot_U;
        PulseDO DO_rot_L;
        PulseDO DO_rot_B;
        PulseDO DO_rot_D;
        MoveL Offs(Target_waiting, 0, 0, -150),v100,fine,Servo;
        PulseDO DO_det;
        PulseDO DO_det_core;
    ENDPROC

    PROC Path_F_2()
        PulseDO DO_att_L;
        PulseDO DO_rot_F;
        PulseDO DO_rot_R;
        PulseDO DO_rot_U;
        PulseDO DO_rot_L;
        PulseDO DO_rot_B;
        PulseDO DO_rot_D;
        MoveL Target_waiting,v100,fine,Servo\WObj:=wobj0;
        PulseDO DO_det;
        PulseDO DO_det_core;
        PulseDO DO_reset;
    ENDPROC

    PROC Path_U_1()
        WaitTime 3;
        PulseDO DO_open_L;
        WaitTime 1;
        MoveL Offs(Target_waiting, 0, 80, 0),v100,fine,Servo;
    ENDPROC

    PROC Path_U_2()
        MoveJ Offs(Target_U, 0, 50, 0),v100,z100,Servo;
        MoveL Offs(Target_U, 0, 12, 0),v100,fine,Servo;
        WaitTime 1;
        PulseDO DO_close_L;
        WaitTime 1;
        PulseDO DO_att_L;
        PulseDO DO_rot_U;
        MoveJ Offs(Target_U_rot, 0, 12, 0),v100,fine,Servo;
        PulseDO DO_det;
        PulseDO DO_det_core;
        WaitTime 1;
        PulseDO DO_open_L;
        WaitTime 1;
        MoveL Offs(Target_U, 0, 50, 0),v100,z100,Servo;
        MoveJ Offs(Target_waiting, 0, 80, 0),v100,fine,Servo;
    ENDPROC

    PROC Path_U_3()
        MoveL Target_waiting,v100,fine,Servo\WObj:=wobj0;
        WaitTime 1;
        PulseDO DO_close_L;
        WaitTime 1;
    ENDPROC

    PROC Path_L_1()
        WaitTime 3;
        PulseDO DO_open_L;
        WaitTime 1;
        MoveL Offs(Target_L, 0, 50, 0),v100,z100,Servo;
        MoveL Offs(Target_L, 0, 12, 0),v100,fine,Servo;
        WaitTime 1;
        PulseDO DO_close_L;
        WaitTime 1;
        PulseDO DO_att_L;
        PulseDO DO_rot_L;
        MoveJ Offs(Target_L_rot, 0, 12, 0),v100,fine,Servo;
        PulseDO DO_det;
        PulseDO DO_det_core;
        PulseDO DO_reset;
        WaitTime 1;
        PulseDO DO_open_L;
        WaitTime 1;
        MoveL Offs(Target_L_rot, 0, 50, 0),v100,z100,Servo;
        MoveJ Offs(Target_waiting, 0, 50, 0),v100,fine,Servo;
        MoveL Target_waiting,v100,fine,Servo\WObj:=wobj0;
        WaitTime 1;
        PulseDO DO_close_L;
        WaitTime 1;
    ENDPROC

    PROC Path_B_1()
        WaitTime 3;
        PulseDO DO_open_L;
        WaitTime 1;
        MoveL Offs(Target_waiting, 0, 25, 0),v100,fine,Servo;
    ENDPROC

    PROC Path_B_2()
        MoveJ Offs(Target_B, 0, 0, -35),v100,z100,Servo;
        MoveL Offs(Target_B, 0, 0, -12),v100,fine,Servo;
        WaitTime 1;
        PulseDO DO_close_L;
        WaitTime 1;
        PulseDO DO_att_L;
        PulseDO DO_rot_B;
        MoveJ Offs(Target_B_rot, 0, 0, -12),v100,fine,Servo;
        PulseDO DO_det;
        PulseDO DO_det_core;
        WaitTime 1;
        PulseDO DO_open_L;
        WaitTime 1;
        MoveL Offs(Target_B_rot, 0, 0, -35),v100,z100,Servo;
        MoveJ Offs(Target_waiting, 0, 25, 0),v100,fine,Servo;
    ENDPROC

    PROC Path_B_3()
        MoveL Target_waiting,v100,fine,Servo\WObj:=wobj0;
        WaitTime 1;
        PulseDO DO_close_L;
        WaitTime 1;
    ENDPROC

    PROC Path_D_1()
        WaitTime 3;
        PulseDO DO_open_L;
        WaitTime 1;
        MoveL Offs(Target_waiting, 0, 100, 0),v100,fine,Servo;
    ENDPROC

    PROC Path_D_2()
        MoveJ Offs(Target_D, 0, 50, 0),v100,z100,Servo;
        MoveL Offs(Target_D, 0, 12, 0),v100,fine,Servo;
        WaitTime 1;
        PulseDO DO_close_L;
        WaitTime 1;
        PulseDO DO_att_L;
        PulseDO DO_rot_D;
        MoveL Offs(Target_D_rot, 0, 12, 0),v100,fine,Servo;
        PulseDO DO_det;
        PulseDO DO_det_core;
        WaitTime 1;
        PulseDO DO_open_L;
        WaitTime 1;
        MoveL Offs(Target_D, 0, 50, 0),v100,z100,Servo;
        MoveJ Offs(Target_waiting, 0, 100, 0),v100,fine,Servo;
    ENDPROC

    PROC Path_D_3()
        MoveL Target_waiting,v100,fine,Servo\WObj:=wobj0;
        WaitTime 1;
        PulseDO DO_close_L;
        WaitTime 1;
    ENDPROC
ENDMODULE

--- Backups/Controller_Rubik/SYSPAR/EIO.cfg ---
EIO:CFG_1.0:6:1::
#
SYSSIG_IN:

      -Signal "Collision_Avoidance" -Action "CollAvoidance"
#
INDUSTRIAL_NETWORK:

      -Name "EtherNetIP" -Connection "Private Network"\
      -Label "EtherNet/IP Adapter Network"

      -Name "DeviceNet" -Label "DeviceNet Master/Slave Network" -Address "2"
#
EIO_CROSS:

      -Name "Cross_Signal_Lamp" -Res "Signal_Lamp" -Act1 "DRV1BRAKE"
#
EIO_SIGNAL_SAFELEVEL:

      -Name "FlangePowerSafeLevel" -ActionWhenStartup "Last"
#
DEVICENET_DEVICE:

      -Name "D652_10" -VendorName "ABB Robotics" -ProductName "24 VDC Unit"\
      -Address 10 -ProductCode 26 -DeviceType 7 -ConnectionType "COS"\
      -OutputSize 2 -InputSize 2
#
DEVICENET_INTERNAL_DEVICE:

      -Name "DN_Internal_Device" -VendorName "ABB Robotics"\
      -ProductName "DeviceNet Internal Slave Device"
#
ETHERNETIP_INTERNAL_DEVICE:

      -Name "EN_Internal_Device" -VendorName "ABB Robotics"\
      -ProductName "EtherNet/IP Internal Adapter Device"
#
EIO_SIGNAL:

      -Name "custom_DI_0" -SignalType "DI" -Device "D652_10" -DeviceMap "0"

      -Name "custom_DI_1" -SignalType "DI" -Device "D652_10" -DeviceMap "1"

      -Name "custom_DI_2" -SignalType "DI" -Device "D652_10" -DeviceMap "2"

      -Name "custom_DI_3" -SignalType "DI" -Device "D652_10" -DeviceMap "3"

      -Name "custom_DI_4" -SignalType "DI" -Device "D652_10" -DeviceMap "4"

      -Name "custom_DI_5" -SignalType "DI" -Device "D652_10" -DeviceMap "5"

      -Name "custom_DI_6" -SignalType "DI" -Device "D652_10" -DeviceMap "6"

      -Name "custom_DI_7" -SignalType "DI" -Device "D652_10" -DeviceMap "7"

      -Name "custom_DO_0" -SignalType "DO" -Device "D652_10" -DeviceMap "0"

      -Name "custom_DO_1" -SignalType "DO" -Device "D652_10" -DeviceMap "1"

      -Name "custom_DO_2" -SignalType "DO" -Device "D652_10" -DeviceMap "2"

      -Name "custom_DO_3" -SignalType "DO" -Device "D652_10" -DeviceMap "3"

      -Name "custom_DO_4" -SignalType "DO" -Device "D652_10" -DeviceMap "4"

      -Name "custom_DO_5" -SignalType "DO" -Device "D652_10" -DeviceMap "5"

      -Name "custom_DO_6" -SignalType "DO" -Device "D652_10" -DeviceMap "6"

      -Name "custom_DO_7" -SignalType "DO" -Device "D652_10" -DeviceMap "7"

      -Name "hall_sensor_joint_1" -SignalType "DI" -Device "D652_10"\
      -DeviceMap "8"

      -Name "hall_sensor_joint_2" -SignalType "DI" -Device "D652_10"\
      -DeviceMap "9"

      -Name "hall_sensor_joint_3" -SignalType "DI" -Device "D652_10"\
      -DeviceMap "11"

      -Name "hall_sensor_joint_4" -SignalType "DI" -Device "D652_10"\
      -DeviceMap "12"

      -Name "hall_sensor_joint_5" -SignalType "DI" -Device "D652_10"\
      -DeviceMap "13"

      -Name "hall_sensor_joint_6" -SignalType "DI" -Device "D652_10"\
      -DeviceMap "14"

      -Name "hall_sensor_joint_7" -SignalType "DI" -Device "D652_10"\
      -DeviceMap "10"

      -Name "hall_sensor_24V_ROB_R" -SignalType "DO" -Device "D652_10"\
      -DeviceMap "8"

      -Name "hall_sensor_24V_ROB_L" -SignalType "DO" -Device "D652_10"\
      -DeviceMap "9"

      -Name "flange_24V_ROB_R" -SignalType "DO" -Device "D652_10"\
      -DeviceMap "10" -SafeLevel "FlangePowerSafeLevel"

      -Name "flange_24V_ROB_L" -SignalType "DO" -Device "D652_10"\
      -DeviceMap "11" -SafeLevel "FlangePowerSafeLevel"

      -Name "Signal_Lamp" -SignalType "DO" -Device "D652_10" -DeviceMap "12"

      -Name "Collision_Avoidance" -SignalType "DO" -Access "All" -Default 1

      -Name "DO_initial" -SignalType "DO"

      -Name "DO_reset" -SignalType "DO"

      -Name "DO_rot_F" -SignalType "DO"

      -Name "DO_rot_R" -SignalType "DO"

      -Name "DO_rot_U" -SignalType "DO"

      -Name "DO_rot_L" -SignalType "DO"

      -Name "DO_rot_B" -SignalType "DO"

      -Name "DO_rot_D" -SignalType "DO"

      -Name "DO_det" -SignalType "DO"

      -Name "DO_att_L" -SignalType "DO"

      -Name "DO_att_R" -SignalType "DO"

      -Name "DO_det_core" -SignalType "DO"

      -Name "DO_open_L" -SignalType "DO"

      -Name "DO_open_R" -SignalType "DO"

      -Name "DO_close_R" -SignalType "DO"

      -Name "DO_close_L" -SignalType "DO"

      -Name "DO_rdy_R" -SignalType "DO"

      -Name "DO_rdy_L" -SignalType "DO"
